{attribute 'qualified_only'}
{attribute 'to_string'}
//{attribute 'strict'}
TYPE TaskA26 :
(
	IDLE,
	PICK_SPACER,
	MEASURE,
	
	size
);
END_TYPE

(* stored: Version 1.1.0.1, ProductVersion 3.1.4024.11
   DUT TaskA26: Id {85428761-490e-4a83-93dc-c714144a7672} *)
